(* CODESYS project mobject-errors.library
   Company: mobject
   DefaultNamespace: mobject-errors
   Version: 0.3.0
   Placeholder: mobject-errors
   Author: mobject dev team
   Title: mobject-errors

Project tree, tasks and I/O mapping:
  libraries: mobject-disposable, 1.1.1 (mobject); mobject-serialization, 0.5.0 (mobject); Tc2_System, * (Beckhoff Automation GmbH)
  Errors/
    function block Error [ST]: OnSerialize, Accept, ErrorType, IsSameAs, Message, SerializeWith
    function block NullError [ST]: ErrorType, Message, SerializeWith
  Interfaces/
    interface I_Error: Accept, ErrorType, IsSameAs, Message
    interface I_ErrorVisitor: VisitError
*)

// Errors/Error
{attribute 'linkalways'} 
{attribute 'no_explicit_call' := 'This FB is a CLASS and must be accessed using methods or properties'}
{attribute 'enable_dynamic_creation'}
FUNCTION_BLOCK ABSTRACT Error EXTENDS Disposable IMPLEMENTS I_Error
VAR
END_VAR

METHOD PROTECTED OnSerialize
VAR_INPUT
	Serializer : I_Serializer;
END_VAR
END_METHOD

METHOD PUBLIC Accept
VAR_INPUT
	Visitor : I_ErrorVisitor;
END_VAR
Visitor.VisitError(THIS^);
END_METHOD

PROPERTY PUBLIC ABSTRACT ErrorType : T_MAXSTRING
GET
END_GET
END_PROPERTY

METHOD PUBLIC IsSameAs : BOOL
VAR_INPUT
	Error : I_Error;
END_VAR
IF Error = 0 THEN
	RETURN;
END_IF

IF Error.ErrorType <> THIS^.ErrorType THEN
	RETURN;
END_IF

IsSameAs := TRUE;
END_METHOD

PROPERTY PUBLIC ABSTRACT Message : T_MAXSTRING
GET
END_GET
END_PROPERTY

METHOD PUBLIC SerializeWith
VAR_INPUT
	Serializer : I_Serializer;
END_VAR
Serializer.StartObject();
Serializer.AddKeyString('errorType',ErrorType);
Serializer.AddKeyString('message',Message);
OnSerialize(Serializer);
Serializer.EndObject();
END_METHOD

END_FUNCTION_BLOCK

// Interfaces/I_Error
INTERFACE I_Error EXTENDS I_Serializable, I_Disposable

METHOD PUBLIC Accept
VAR_INPUT
	Visitor : I_ErrorVisitor;
END_VAR
END_METHOD

PROPERTY ErrorType : T_MAXSTRING
GET
END_GET
END_PROPERTY

METHOD PUBLIC IsSameAs : BOOL
VAR_INPUT
	Error : I_Error;
END_VAR
END_METHOD

PROPERTY Message : T_MAXSTRING
GET
END_GET
END_PROPERTY

END_INTERFACE

// Interfaces/I_ErrorVisitor
INTERFACE I_ErrorVisitor

METHOD VisitError
VAR_INPUT
	VisitingError : I_Error;
END_VAR
END_METHOD

END_INTERFACE

// Errors/NullError
{attribute 'linkalways'} 
{attribute 'no_explicit_call' := 'This FB is a CLASS and must be accessed using methods or properties'}
{attribute 'enable_dynamic_creation'}
FUNCTION_BLOCK NullError EXTENDS Error
VAR
END_VAR

PROPERTY ErrorType : T_MAXSTRING
GET
END_GET
END_PROPERTY

PROPERTY PUBLIC Message : T_MAXSTRING
GET
END_GET
END_PROPERTY

METHOD PUBLIC SerializeWith
VAR_INPUT
	Serializer : I_Serializer;
END_VAR
END_METHOD

END_FUNCTION_BLOCK
